{attribute 'linkalways'} 
{attribute 'no_explicit_call' := 'This FB is a CLASS and must be accessed using methods or properties'}
{attribute 'enable_dynamic_creation'}
FUNCTION_BLOCK FINAL SUB_USINT EXTENDS Node
VAR
	in1 : _USINT(0);
	in2 : _USINT(0);
	out : _USINT(0);
END_VAR

METHOD PUBLIC Clone : I_Node
VAR
	pNode : POINTER TO SUB_USINT;
END_VAR
pNode := __NEW(SUB_USINT);
Clone := pNode^;
END_METHOD

METHOD FB_init : BOOL
VAR_INPUT
	bInitRetains : BOOL; // if TRUE, the retain variables are initialized (warm start / cold start)
	bInCopyCode : BOOL;  // if TRUE, the instance afterwards gets moved into the copy code (online change)
END_VAR
AddInput('in1',THIS^.in1);
AddInput('in2',THIS^.in2);
AddOutput('out', THIS^.out);
END_METHOD

METHOD PROTECTED OnExecute
VAR
END_VAR
out.Value := in1.Value - in2.Value;
END_METHOD

END_FUNCTION_BLOCK

(* stored: Version 1.1.0.1, ProductVersion 3.1.4024.15
   POU SUB_USINT: Id {828d58f9-b1b8-4ed3-9ddf-8d6a192fbf44}, SpecialFunc None
   Folder Constructor: Id {b288d1bf-9962-4c21-a198-eb4898843021}
   Method Clone: Id {daebed2b-2cee-49b9-8187-80da20975177}
   Method FB_init: Id {23f9e7ca-c770-4238-866b-30a38bc984db}
   Method OnExecute: Id {a5044592-e7e8-45c3-a88d-ee4333cfe57f} *)
